// SIMATIC S7-200 SMART project (STEP 7-Micro/WIN SMART), CPU SR20

ORGANIZATION_BLOCK MAIN:OB1
TITLE=Program Comments
BEGIN
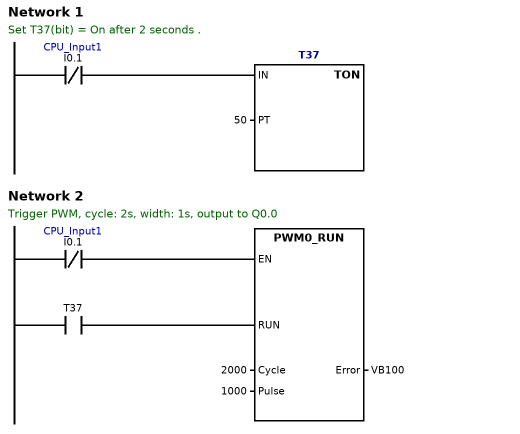
Network 1
// Set T37(bit) = On after 2 seconds .
// (network saved uncompiled; LAD cells follow)
// row 0: c0 -|/|- CPU_Input1:I0.1  c1 --  c2 [TON T37 IN:=power@row0, PT:=50]
// row 1: c2 [box]
Network 2
// Trigger PWM, cycle: 2s, width: 1s, output to Q0.0
LDN    CPU_Input1:I0.1
=      L60.0
LD     T37
=      L63.7
LD     L60.0
CALL   PWM0_RUN:SBR1, L63.7, 2000, 1000, VB100
END_ORGANIZATION_BLOCK

SUBROUTINE_BLOCK SBR_0:SBR0
TITLE=Subroutine Comments
BEGIN
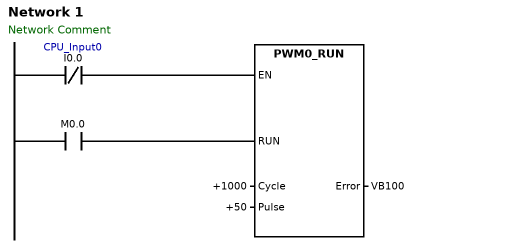
Network 1
// Network Comment
LDN    CPU_Input0:I0.0
=      L60.0
LD     M0.0
=      L63.7
LD     L60.0
CALL   PWM0_RUN:SBR1, L63.7, +1000, +50, VB100
END_SUBROUTINE_BLOCK

// SBR1: protected block, not included
